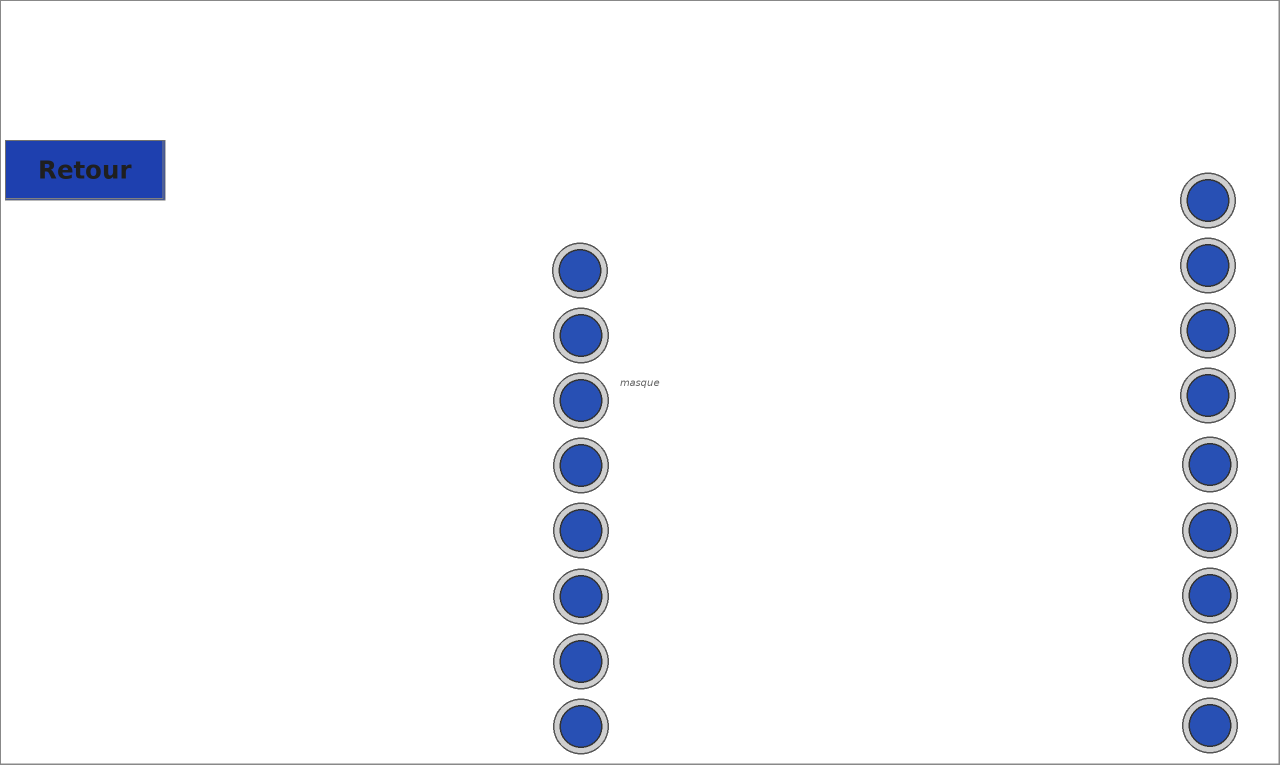
VISUALIZATION Maintenance_7  // 1280x765
    Frame (0,0 1280x765)
        shows masque()
    Rectangle (284,73 232x40), "Etats des E/S TOR"
    Button (5,140 160x60), "Retour", invisible if: Mode_Cabine_Depollution
        OnMouseDown: execute {
            IF (Option_Com_RegSouf_Ultrason)
            	THEN
            		VisuElems.CURRENTVISU := 'Maintenance_6';
            	ELSIF (Option_Cabine_Climatique)
            		THEN
            		VisuElems.CURRENTVISU := 'Maintenance_5';
            	ELSIF (Option_WC_GV OR Option_WC_PV OR Option_Prise)
            		THEN
            		VisuElems.CURRENTVISU := 'Maintenance_4';
            	ELSIF (Option_Bas_Debit OR Option_Douchette OR Option_NEP)
            		THEN
            		VisuElems.CURRENTVISU := 'Maintenance_3';
            	ELSIF (Option_Douche OR Option_Lavabo)
            		THEN
            		VisuElems.CURRENTVISU := 'Maintenance_2';
            	ELSIF (Option_RegSouf_Ultrason OR Option_Reg_Etanche_Ext OR Option_V3V_EauMitig)
            		THEN
            		VisuElems.CURRENTVISU := 'Maintenance_1';
            	ELSE
            	VisuElems.CURRENTVISU := 'menu';
            END_IF
        }
    Rectangle (7,238 533x65), "ETOR1_Fdc_Va_Vid_Lavabo_Ouv"
    Rectangle (9,303 533x65), "ETOR2_Fdc_Va_Vid_Lavabo_Ferm"
    Rectangle (7,368 533x65), "ETOR3_Info_Ma_Prise"
    Rectangle (7,433 533x65), "ETOR4_Service_Humi_CTA"
    Rectangle (7,498 533x65), "ETOR5_Def_Humi_CTA"
    Rectangle (7,564 533x65), "ETOR6_Info_Contact_Porte"
    Rectangle (7,629 533x65), "ETOR7_Def_MotRep_Souf_CTA"
    Rectangle (7,694 533x65), "ETOR8_Def_MotSouf_Souf_CTA"
    Rectangle (637,432 533x65), "ETOR13_Marche_BatElec_CTA"
    Rectangle (637,498 533x65), "STOR1_Cmd_EV_Alim_Lavabo"
    Rectangle (637,563 533x65), "STOR2_Cmd_Va_Vid_Lavabo"
    Rectangle (637,628 533x65), "STOR3_Cmd_Ma_Prise"
    Rectangle (637,693 533x65), "STOR4_Cmd_BatElec_CTA"
    Lamp1 (548,238 64x65), variable: ETOR1_Fdc_Va_Vid_Lavabo_Ouv, style: Lamp-Lamp1-Blue
    Lamp1 (549,303 64x65), variable: ETOR2_Fdc_Va_Vid_Lavabo_Ferm, style: Lamp-Lamp1-Blue
    Lamp1 (549,368 64x65), variable: ETOR3_Info_Ma_Prise, style: Lamp-Lamp1-Blue
    Lamp1 (549,433 64x65), variable: ETOR4_Service_Humi_CTA, style: Lamp-Lamp1-Blue
    Lamp1 (549,498 64x65), variable: ETOR5_Def_Humi_CTA, style: Lamp-Lamp1-Blue
    Lamp1 (549,564 64x65), variable: ETOR6_Info_Contact_Porte, style: Lamp-Lamp1-Blue
    Lamp1 (549,629 64x65), variable: ETOR7_Def_MotRep_Souf_CTA, style: Lamp-Lamp1-Blue
    Lamp1 (549,694 64x65), variable: ETOR8_Def_MotSouf_Souf_CTA, style: Lamp-Lamp1-Blue
    Lamp1 (1178,432 64x65), variable: ETOR13_Marche_BatElec_CTA, style: Lamp-Lamp1-Blue
    Lamp1 (1178,498 64x65), variable: STOR1_Cmd_EV_Alim_Lavabo, style: Lamp-Lamp1-Blue
    Lamp1 (1178,563 64x65), variable: STOR2_Cmd_Va_Vid_Lavabo, style: Lamp-Lamp1-Blue
    Lamp1 (1178,628 64x65), variable: STOR3_Cmd_Ma_Prise, style: Lamp-Lamp1-Blue
    Lamp1 (1178,693 64x65), variable: STOR4_Cmd_BatElec_CTA, style: Lamp-Lamp1-Blue
    Rectangle (635,168 533x65), "ETOR9_Def_Alim_BatElec_CTA"
    Lamp1 (1176,168 64x65), variable: ETOR9_Def_Alim_BatElec_CTA, style: Lamp-Lamp1-Blue
    Rectangle (635,233 533x65), "ETOR10_Hygrostat_Souf_CT"
    Lamp1 (1176,233 64x65), variable: ETOR10_Hygrostat_Souf_CT, style: Lamp-Lamp1-Blue
    Rectangle (635,298 533x65), "ETOR11_Pressostat_Secu"
    Lamp1 (1176,298 64x65), variable: ETOR11_Pressostat_Secu, style: Lamp-Lamp1-Blue
    Rectangle (635,363 533x65), "ETOR12_Thermostat_Secu"
    Lamp1 (1176,363 64x65), variable: ETOR12_Thermostat_Secu, style: Lamp-Lamp1-Blue
END_VISUALIZATION

(* stored: Version 1.1.0.1, ProductVersion 3.1.4024.16
   Visu Maintenance_7: Id {ff041f17-9306-4d80-ab6c-93296337fc73} *)
